PROGRAM SP2_1_Y120
VAR
	CompareOutput120_00: CMP_OC_DW;
	CompareOutput120_01: CMP_OC_DW;
	CompareOutput120_02: CMP_OC_DW;
	CompareOutput120_03: CMP_OC_DW;
	CompareOutput120_04: CMP_OC_DW;
	CompareOutput120_05: CMP_OC_DW;
	CompareOutput120_06: CMP_OC_DW;
	CompareOutput120_07: CMP_OC_DW;
	CompareOutput120_08: CMP_OC_DW;
	CompareOutput120_09: CMP_OC_DW;
	CompareOutput120_10: CMP_OC_DW;
	CompareOutput120_11: CMP_OC_DW;
	CompareOutput120_12: CMP_OC_DW;
	CompareOutput120_13: CMP_OC_DW;
	CompareOutput120_14: CMP_OC_DW;
	CompareOutput120_15: CMP_OC_DW;

END_VAR

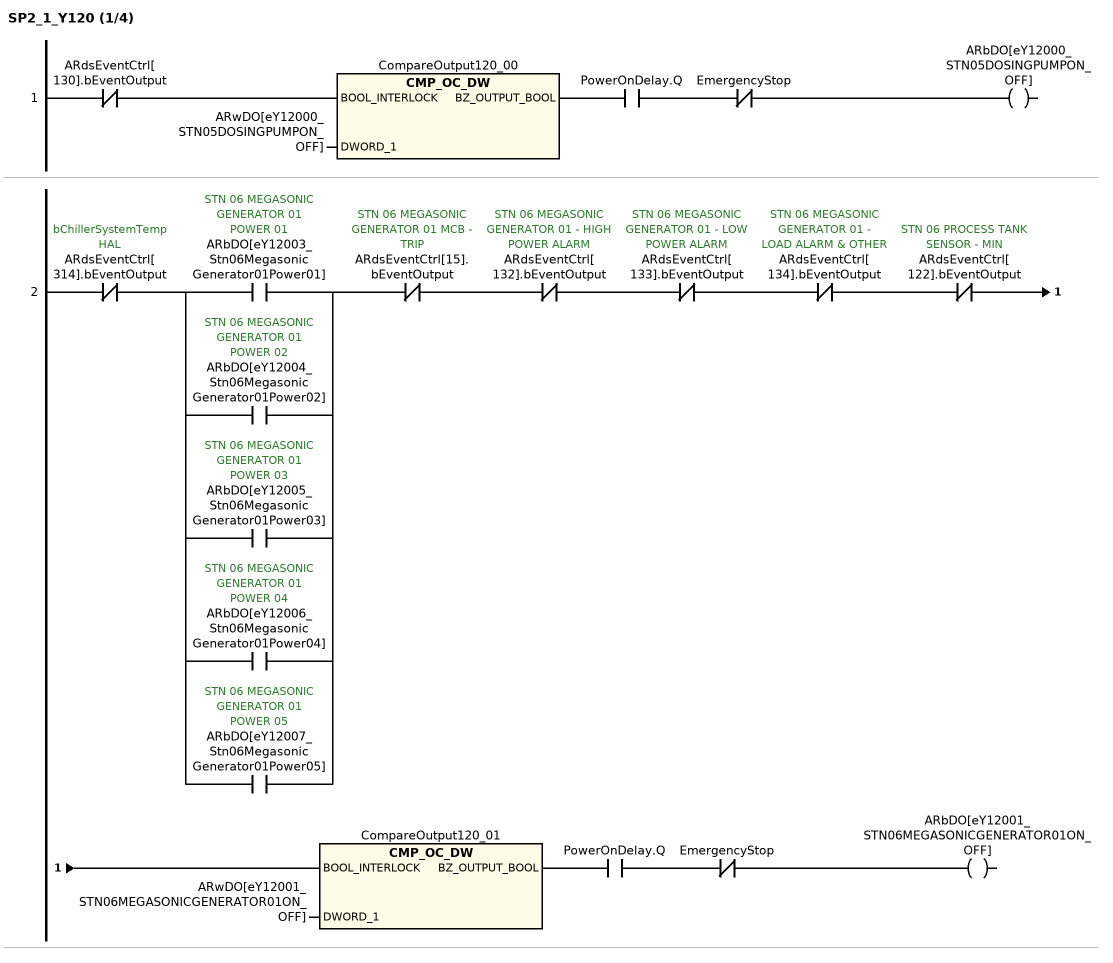
// NETWORK 1
CompareOutput120_00(BOOL_INTERLOCK := NOT ARdsEventCtrl[130].bEventOutput, DWORD_1 := ARwDO[eY12000_STN05DOSINGPUMPON_OFF]); // CMP_OC_DW
ARbDO[eY12000_STN05DOSINGPUMPON_OFF] := CompareOutput120_00.BZ_OUTPUT_BOOL AND PowerOnDelay.Q AND NOT EmergencyStop;

// NETWORK 2
//   ARdsEventCtrl[314].bEventOutput: bChillerSystemTempHAL
//   ARbDO[eY12003_Stn06MegasonicGenerator01Power01]: STN 06 MEGASONIC GENERATOR 01 POWER 01
//   ARbDO[eY12004_Stn06MegasonicGenerator01Power02]: STN 06 MEGASONIC GENERATOR 01 POWER 02
//   ARbDO[eY12005_Stn06MegasonicGenerator01Power03]: STN 06 MEGASONIC GENERATOR 01 POWER 03
//   ARbDO[eY12006_Stn06MegasonicGenerator01Power04]: STN 06 MEGASONIC GENERATOR 01 POWER 04
//   ARbDO[eY12007_Stn06MegasonicGenerator01Power05]: STN 06 MEGASONIC GENERATOR 01 POWER 05
//   ARdsEventCtrl[15].bEventOutput: STN 06 MEGASONIC GENERATOR 01 MCB - TRIP
//   ARdsEventCtrl[132].bEventOutput: STN 06 MEGASONIC GENERATOR 01 - HIGH POWER ALARM
//   ARdsEventCtrl[133].bEventOutput: STN 06 MEGASONIC GENERATOR 01 - LOW POWER ALARM
//   ARdsEventCtrl[134].bEventOutput: STN 06 MEGASONIC GENERATOR 01 - LOAD ALARM & OTHER
//   ARdsEventCtrl[122].bEventOutput: STN 06 PROCESS TANK SENSOR - MIN
CompareOutput120_01(BOOL_INTERLOCK := NOT ARdsEventCtrl[314].bEventOutput AND (ARbDO[eY12003_Stn06MegasonicGenerator01Power01] OR ARbDO[eY12004_Stn06MegasonicGenerator01Power02] OR ARbDO[eY12005_Stn06MegasonicGenerator01Power03] OR ARbDO[eY12006_Stn06MegasonicGenerator01Power04] OR ARbDO[eY12007_Stn06MegasonicGenerator01Power05]) AND NOT ARdsEventCtrl[15].bEventOutput AND NOT ARdsEventCtrl[132].bEventOutput AND NOT ARdsEventCtrl[133].bEventOutput AND NOT ARdsEventCtrl[134].bEventOutput AND NOT ARdsEventCtrl[122].bEventOutput, DWORD_1 := ARwDO[eY12001_STN06MEGASONICGENERATOR01ON_OFF]); // CMP_OC_DW
ARbDO[eY12001_STN06MEGASONICGENERATOR01ON_OFF] := CompareOutput120_01.BZ_OUTPUT_BOOL AND PowerOnDelay.Q AND NOT EmergencyStop;

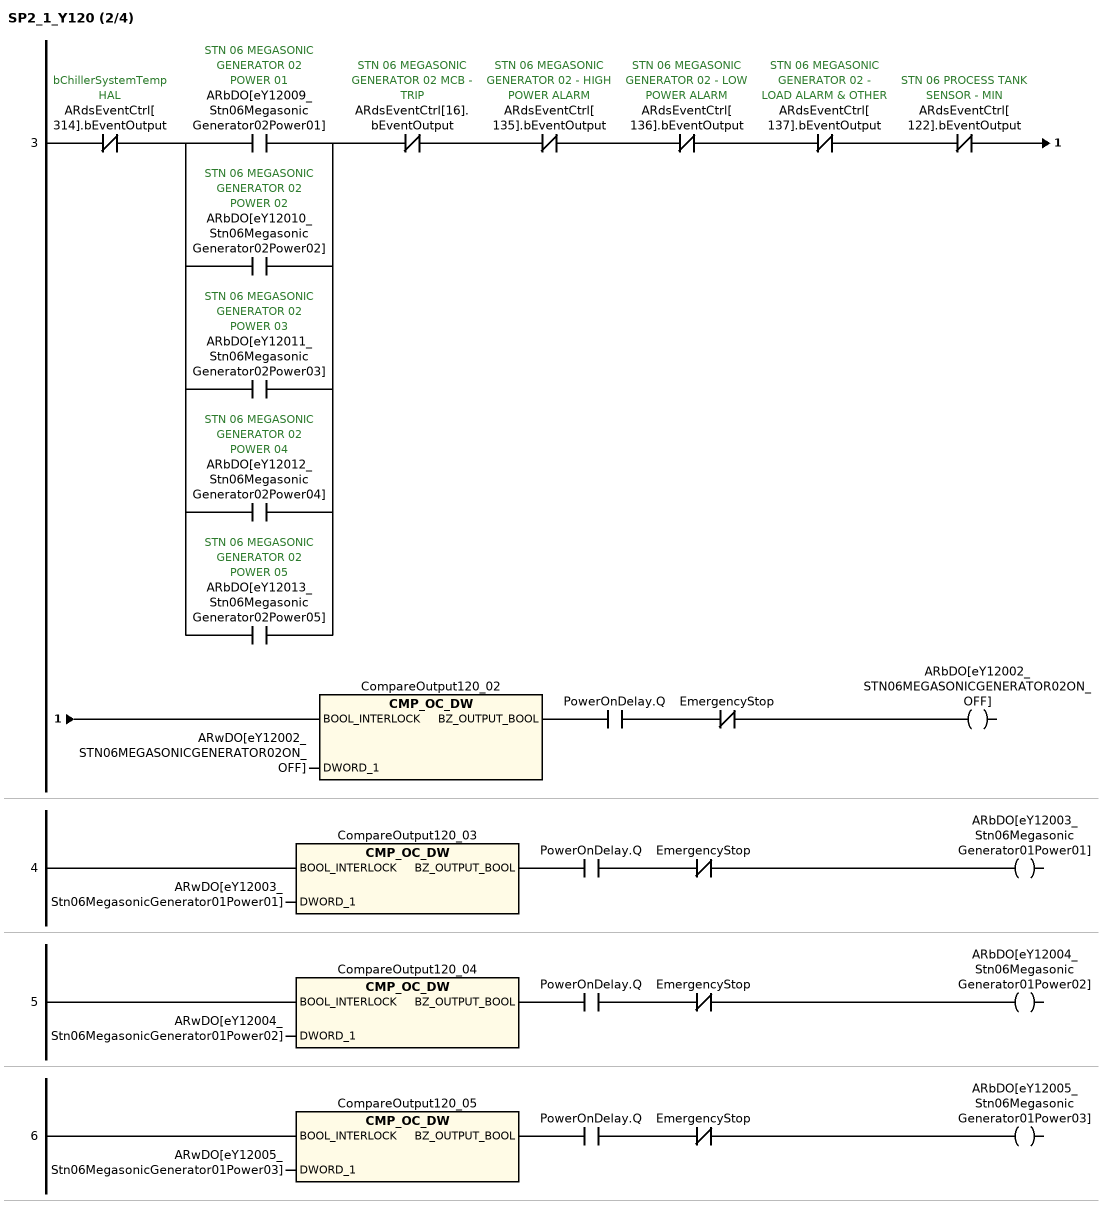
// NETWORK 3
//   ARdsEventCtrl[314].bEventOutput: bChillerSystemTempHAL
//   ARbDO[eY12009_Stn06MegasonicGenerator02Power01]: STN 06 MEGASONIC GENERATOR 02 POWER 01
//   ARbDO[eY12010_Stn06MegasonicGenerator02Power02]: STN 06 MEGASONIC GENERATOR 02 POWER 02
//   ARbDO[eY12011_Stn06MegasonicGenerator02Power03]: STN 06 MEGASONIC GENERATOR 02 POWER 03
//   ARbDO[eY12012_Stn06MegasonicGenerator02Power04]: STN 06 MEGASONIC GENERATOR 02 POWER 04
//   ARbDO[eY12013_Stn06MegasonicGenerator02Power05]: STN 06 MEGASONIC GENERATOR 02 POWER 05
//   ARdsEventCtrl[16].bEventOutput: STN 06 MEGASONIC GENERATOR 02 MCB - TRIP
//   ARdsEventCtrl[135].bEventOutput: STN 06 MEGASONIC GENERATOR 02 - HIGH POWER ALARM
//   ARdsEventCtrl[136].bEventOutput: STN 06 MEGASONIC GENERATOR 02 - LOW POWER ALARM
//   ARdsEventCtrl[137].bEventOutput: STN 06 MEGASONIC GENERATOR 02 - LOAD ALARM & OTHER
//   ARdsEventCtrl[122].bEventOutput: STN 06 PROCESS TANK SENSOR - MIN
CompareOutput120_02(BOOL_INTERLOCK := NOT ARdsEventCtrl[314].bEventOutput AND (ARbDO[eY12009_Stn06MegasonicGenerator02Power01] OR ARbDO[eY12010_Stn06MegasonicGenerator02Power02] OR ARbDO[eY12011_Stn06MegasonicGenerator02Power03] OR ARbDO[eY12012_Stn06MegasonicGenerator02Power04] OR ARbDO[eY12013_Stn06MegasonicGenerator02Power05]) AND NOT ARdsEventCtrl[16].bEventOutput AND NOT ARdsEventCtrl[135].bEventOutput AND NOT ARdsEventCtrl[136].bEventOutput AND NOT ARdsEventCtrl[137].bEventOutput AND NOT ARdsEventCtrl[122].bEventOutput, DWORD_1 := ARwDO[eY12002_STN06MEGASONICGENERATOR02ON_OFF]); // CMP_OC_DW
ARbDO[eY12002_STN06MEGASONICGENERATOR02ON_OFF] := CompareOutput120_02.BZ_OUTPUT_BOOL AND PowerOnDelay.Q AND NOT EmergencyStop;

// NETWORK 4
CompareOutput120_03(BOOL_INTERLOCK := TRUE, DWORD_1 := ARwDO[eY12003_Stn06MegasonicGenerator01Power01]); // CMP_OC_DW
ARbDO[eY12003_Stn06MegasonicGenerator01Power01] := CompareOutput120_03.BZ_OUTPUT_BOOL AND PowerOnDelay.Q AND NOT EmergencyStop;

// NETWORK 5
CompareOutput120_04(BOOL_INTERLOCK := TRUE, DWORD_1 := ARwDO[eY12004_Stn06MegasonicGenerator01Power02]); // CMP_OC_DW
ARbDO[eY12004_Stn06MegasonicGenerator01Power02] := CompareOutput120_04.BZ_OUTPUT_BOOL AND PowerOnDelay.Q AND NOT EmergencyStop;

// NETWORK 6
CompareOutput120_05(BOOL_INTERLOCK := TRUE, DWORD_1 := ARwDO[eY12005_Stn06MegasonicGenerator01Power03]); // CMP_OC_DW
ARbDO[eY12005_Stn06MegasonicGenerator01Power03] := CompareOutput120_05.BZ_OUTPUT_BOOL AND PowerOnDelay.Q AND NOT EmergencyStop;

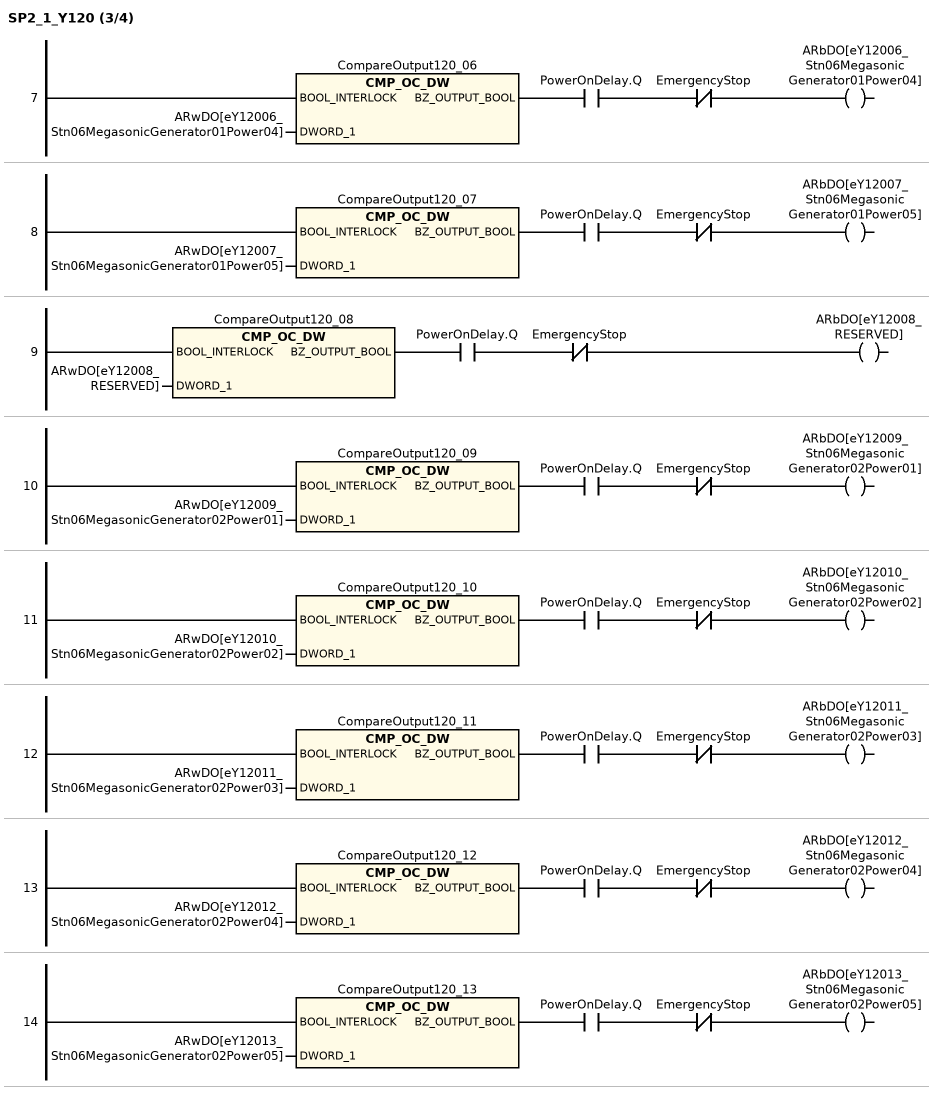
// NETWORK 7
CompareOutput120_06(BOOL_INTERLOCK := TRUE, DWORD_1 := ARwDO[eY12006_Stn06MegasonicGenerator01Power04]); // CMP_OC_DW
ARbDO[eY12006_Stn06MegasonicGenerator01Power04] := CompareOutput120_06.BZ_OUTPUT_BOOL AND PowerOnDelay.Q AND NOT EmergencyStop;

// NETWORK 8
CompareOutput120_07(BOOL_INTERLOCK := TRUE, DWORD_1 := ARwDO[eY12007_Stn06MegasonicGenerator01Power05]); // CMP_OC_DW
ARbDO[eY12007_Stn06MegasonicGenerator01Power05] := CompareOutput120_07.BZ_OUTPUT_BOOL AND PowerOnDelay.Q AND NOT EmergencyStop;

// NETWORK 9
CompareOutput120_08(BOOL_INTERLOCK := TRUE, DWORD_1 := ARwDO[eY12008_RESERVED]); // CMP_OC_DW
ARbDO[eY12008_RESERVED] := CompareOutput120_08.BZ_OUTPUT_BOOL AND PowerOnDelay.Q AND NOT EmergencyStop;

// NETWORK 10
CompareOutput120_09(BOOL_INTERLOCK := TRUE, DWORD_1 := ARwDO[eY12009_Stn06MegasonicGenerator02Power01]); // CMP_OC_DW
ARbDO[eY12009_Stn06MegasonicGenerator02Power01] := CompareOutput120_09.BZ_OUTPUT_BOOL AND PowerOnDelay.Q AND NOT EmergencyStop;

// NETWORK 11
CompareOutput120_10(BOOL_INTERLOCK := TRUE, DWORD_1 := ARwDO[eY12010_Stn06MegasonicGenerator02Power02]); // CMP_OC_DW
ARbDO[eY12010_Stn06MegasonicGenerator02Power02] := CompareOutput120_10.BZ_OUTPUT_BOOL AND PowerOnDelay.Q AND NOT EmergencyStop;

// NETWORK 12
CompareOutput120_11(BOOL_INTERLOCK := TRUE, DWORD_1 := ARwDO[eY12011_Stn06MegasonicGenerator02Power03]); // CMP_OC_DW
ARbDO[eY12011_Stn06MegasonicGenerator02Power03] := CompareOutput120_11.BZ_OUTPUT_BOOL AND PowerOnDelay.Q AND NOT EmergencyStop;

// NETWORK 13
CompareOutput120_12(BOOL_INTERLOCK := TRUE, DWORD_1 := ARwDO[eY12012_Stn06MegasonicGenerator02Power04]); // CMP_OC_DW
ARbDO[eY12012_Stn06MegasonicGenerator02Power04] := CompareOutput120_12.BZ_OUTPUT_BOOL AND PowerOnDelay.Q AND NOT EmergencyStop;

// NETWORK 14
CompareOutput120_13(BOOL_INTERLOCK := TRUE, DWORD_1 := ARwDO[eY12013_Stn06MegasonicGenerator02Power05]); // CMP_OC_DW
ARbDO[eY12013_Stn06MegasonicGenerator02Power05] := CompareOutput120_13.BZ_OUTPUT_BOOL AND PowerOnDelay.Q AND NOT EmergencyStop;

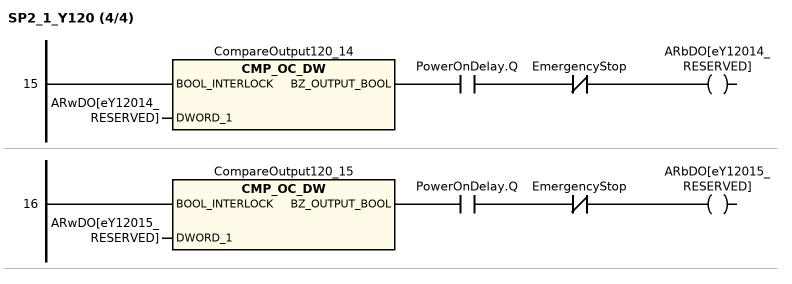
// NETWORK 15
CompareOutput120_14(BOOL_INTERLOCK := TRUE, DWORD_1 := ARwDO[eY12014_RESERVED]); // CMP_OC_DW
ARbDO[eY12014_RESERVED] := CompareOutput120_14.BZ_OUTPUT_BOOL AND PowerOnDelay.Q AND NOT EmergencyStop;

// NETWORK 16
CompareOutput120_15(BOOL_INTERLOCK := TRUE, DWORD_1 := ARwDO[eY12015_RESERVED]); // CMP_OC_DW
ARbDO[eY12015_RESERVED] := CompareOutput120_15.BZ_OUTPUT_BOOL AND PowerOnDelay.Q AND NOT EmergencyStop;

END_PROGRAM

(* stored: Version 1.1.0.1, ProductVersion 3.1.4024.11
   POU SP2_1_Y120: Id {2e179fdd-972e-4fbb-b09b-c81dd1dc096e}, SpecialFunc None *)
